// TIA Portal project "Water Fountain Sequence" (V17)
// Water Fountain Sequence
// The fountain should operate in three stages.
// High spray for 15 sec
// Low spray for 10 sec
// OFF for 5 sec

(* hardware
DEVICE "S7-1200 station_1"  S7-1200 Station
   slot 0: "Rack_0"  S7-1200 Rack  Rack  V1.0
   slot 1: "PLC_1"  CPU 1212C AC/DC/Rly  6ES7 212-1BE40-0XB0  V4.5
*)

// ===== PLC "PLC_1"  CPU 1212C AC/DC/Rly =====

VAR_GLOBAL   // PLC tag table "Default tag table"
   "Start_fountain" AT %I0.0 : Bool;
   "Stop_system" AT %I0.1 : Bool;
   "High_spray" AT %Q0.0 : Bool;
   "Low_spray" AT %Q0.1 : Bool;
   "Fountain" AT %M0.0 : Bool;
   "Tag_1" AT %M0.1 : Bool;
END_VAR

// folder: System blocks/Program resources

DATA_BLOCK "IEC_Timer_0_DB"   // DB1
{ S7_Optimized_Access := 'TRUE' }
AUTHOR : Simatic
FAMILY : IEC
NAME : IEC_TMR
VERSION : 1.0
// stored: InstanceOfName IEC_TIMER
"IEC_TIMER"
BEGIN
END_DATA_BLOCK

DATA_BLOCK "IEC_Timer_0_DB_1"   // DB2
{ S7_Optimized_Access := 'TRUE' }
AUTHOR : Simatic
FAMILY : IEC
NAME : IEC_TMR
VERSION : 1.0
// stored: InstanceOfName IEC_TIMER
"IEC_TIMER"
BEGIN
END_DATA_BLOCK

DATA_BLOCK "IEC_Timer_0_DB_2"   // DB3
{ S7_Optimized_Access := 'TRUE' }
AUTHOR : Simatic
FAMILY : IEC
NAME : IEC_TMR
VERSION : 1.0
// stored: InstanceOfName IEC_TIMER
"IEC_TIMER"
BEGIN
END_DATA_BLOCK

// folder: (top level)

ORGANIZATION_BLOCK "Main"   // OB1, LAD, ProgramCycle
TITLE = "Main Program Sweep (Cycle)"
{ S7_Optimized_Access := 'TRUE' }
VERSION : 0.1
   VAR_INPUT
      Initial_Call : Bool;   // Initial call of this OB
      Remanence : Bool;   // =True, if remanent data are available
   END_VAR
   VAR_TEMP   // added for the SCL form of the ladder/FBD networks
      _w1 : Bool;
   END_VAR
BEGIN

REGION Network 1
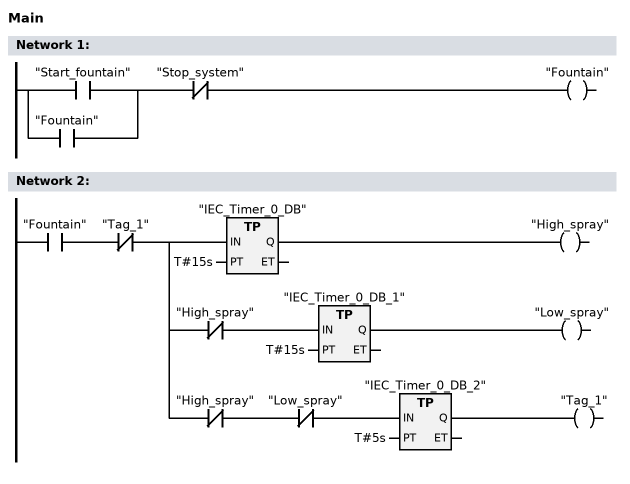
   RUNG wire#powerrail
      Contact( "Start_fountain" )
      wire#w1
      I_Contact( "Stop_system" )
      Coil( "Fountain" )
   END_RUNG
   RUNG wire#powerrail
      Contact( "Fountain" )
   END_RUNG wire#w1
   // the same network as SCL:
   "Fountain" := ("Start_fountain" OR "Fountain") AND NOT "Stop_system";
END_REGION

REGION Network 2
   #_w1 := "Fountain" AND NOT "Tag_1";
   "IEC_Timer_0_DB".TP(IN := #_w1, PT := T#15s);
   "High_spray" := "IEC_Timer_0_DB".Q;
   "IEC_Timer_0_DB_1".TP(IN := #_w1 AND NOT "High_spray", PT := T#15s);
   "Low_spray" := "IEC_Timer_0_DB_1".Q;
   "IEC_Timer_0_DB_2".TP(IN := #_w1 AND NOT "High_spray" AND NOT "Low_spray", PT := T#5s);
   "Tag_1" := "IEC_Timer_0_DB_2".Q;
END_REGION
END_ORGANIZATION_BLOCK